FUNCTION_BLOCK FB_Counter

VAR
	vdiCounterValue : DINT;
END_VAR

METHOD M_AddCounterValue
VAR
END_VAR
vdiCounterValue := vdiCounterValue + 1;
END_METHOD

END_FUNCTION_BLOCK

(* stored: Version 1.1.0.1, ProductVersion 3.1.4024.9
   POU FB_Counter: Id {fb7c3b3d-8d82-4d2d-a702-d92db386dd1f}, SpecialFunc None
   Method M_AddCounterValue: Id {8b473c10-0a6a-4c5d-8d38-555b2241fc26} *)
